ABB RAPID module: Wobj_wobj1eSergiox21.MOD

MODULE Wobj_wobj1eSergiox21
	! Points are read in order of declaration.
  ! Please do not change the order of points!

  LOCAL PERS robtarget pWobj_O_PointX1:=[[-459.0601,-408.0227,308.6543],[0.277203530073166,0.314697861671448,-0.90715229511261,-0.034614447504282],[-2,-1,2,0],[9E+09,9E+09,9E+09,9E+09,9E+09,9E+09]];
	LOCAL PERS robtarget pWobj_O_PointX2:=[[-605.9445,-418.088,319.2509],[0.277176558971405,0.314687937498093,-0.907163679599762,-0.0346214137971401],[-2,-1,2,0],[9E+09,9E+09,9E+09,9E+09,9E+09,9E+09]];
	LOCAL PERS robtarget pWobj_O_PointY1:=[[-483.3394,-40.16927,308.2043],[0.277250319719315,0.314726442098618,-0.907128632068634,-0.0346000455319881],[-2,0,1,0],[9E+09,9E+09,9E+09,9E+09,9E+09,9E+09]];

ENDMODULE
